FUNCTION_BLOCK FB_Base IMPLEMENTS I_Base
VAR_INPUT
END_VAR
VAR_OUTPUT
END_VAR
VAR
	{attribute 'instance-path'} 
    {attribute 'noinit'}
    {attribute 'hide'} 
    sInstancePath:		STRING(255);
	eState: 			E_Base;
	eRequest: 			E_Base;
	nState: 			INT;
	sName:				STRING(255):= 'test-run'; 	// Name OF the entire test run
	sTimestamp:			STRING(39);						// timestamp   Date and time of when the test suite was executed (in ISO 8601 format)
    {attribute 'hide'} 
	fbTask:				GETCURTASKINDEX;
	fbGetTime:			NT_GetTime;
	fCycleTime: 		LREAL;	
END_VAR

fbGetTime();

CASE eState OF
	E_Base.Init:
		IF M_Init() THEN
			eState:= E_Base.Stopped;
			nState:= 0;
		END_IF
		
	E_Base.Stopped:
		IF M_Stopped() THEN
			eState:= E_Base.Starting;
			nState:= 0;
		ELSE
			CASE eRequest OF
				E_Base.Starting, E_Base.Started:
					eState:= E_Base.Starting;
					nState:= 0;
			END_CASE
		END_IF
		
	E_Base.Starting:
		IF M_Starting() THEN
			eState:= E_Base.Started;
			nState:= 0;
		ELSE
			CASE eRequest OF
				E_Base.Started:
					eState:= E_Base.Started;
					nState:= 0;
			END_CASE
		END_IF
		
	E_Base.Started:
		IF M_Started() THEN
			eState:= E_Base.Stopping;
			nState:= 0;
		ELSE
			CASE eRequest OF
				E_Base.Stopping, E_Base.Stopped:
					eState:= E_Base.Stopping;
					nState:= 0;
			END_CASE
		END_IF
		
	E_Base.Stopping:
		IF M_Stopping() THEN
			eState:= E_Base.Stopped;
			nState:= 0;
		ELSE
			CASE eRequest OF
				E_Base.Stopped:
					eState:= E_Base.Stopped;
					nState:= 0;
			END_CASE
		END_IF
		
END_CASE

eRequest:= eState;

METHOD INTERNAL M_GetName : STRING(255)
VAR_INPUT
	sInstancePath:		STRING(255);
END_VAR
VAR
    sName:				STRING(255);
    nPosition:			INT;
END_VAR
sName := CONCAT(TwinCAT_SystemInfoVarList._AppInfo.ProjectName, '.');

nPosition := FIND(sInstancePath, sName);

IF nPosition > 0 THEN
    M_GetName:= DELETE(sInstancePath, nPosition-1 + LEN(sName), 1);
END_IF

nPosition := FIND(sInstancePath, sName);

IF nPosition > 0 THEN
    M_GetName:= DELETE(M_GetName, nPosition - 1 + LEN(sName), 1);
END_IF

nPosition:= FIND(STR1 := M_GetName, '.');
M_GetName:= RIGHT(STR := M_GetName, LEN(STR := M_GetName) - nPosition);
END_METHOD

METHOD PROTECTED M_Init : BOOL
VAR_INPUT
END_VAR
fbTask();

M_Init:= True;
END_METHOD

METHOD M_Request : BOOL
VAR_INPUT
	eState:		E_Base;
END_VAR
eRequest:= eState;
M_Request:= TRUE;
END_METHOD

METHOD PROTECTED M_Started : BOOL
VAR_INPUT
END_VAR
END_METHOD

METHOD PROTECTED M_Starting : BOOL
VAR_INPUT
END_VAR
IF fbGetTime.START THEN
	IF fbGetTime.BUSY THEN
		;
	ELSE
		sTimestamp:= SYSTEMTIME_TO_ISO8601(fbGetTime.TIMESTR, 0, FALSE, 2);
		fbGetTime.START:= FALSE;
		M_Starting:= TRUE;
	END_IF
ELSE
	sName:= M_GetName(sInstancePath);
	fCycleTime:= UDINT_TO_LREAL(TwinCAT_SystemInfoVarList._TaskInfo[fbTask.index].CycleTime) / 10000000;
	fbGetTime.START:= TRUE;
END_IF
END_METHOD

METHOD PROTECTED M_Stopped : BOOL
VAR_INPUT
END_VAR
END_METHOD

METHOD PROTECTED M_Stopping : BOOL
VAR_INPUT
END_VAR
M_Stopping:= True;
END_METHOD

PROPERTY PUBLIC P_Name : STRING(255)
GET
P_Name:= sName;
END_GET
SET
sName:= P_Name;
END_SET
END_PROPERTY

PROPERTY PUBLIC P_State : E_Base
GET
P_State:= eState;
END_GET
END_PROPERTY

END_FUNCTION_BLOCK

(* stored: Version 1.1.0.1
   POU FB_Base: Id {83180dff-a34f-4cb4-bb72-3f658f1a77bc}, SpecialFunc None
   Method M_GetName: Id {7644e4a6-816c-4e95-a1be-94a500976a8c}
   Method M_Init: Id {e2b264db-76f6-0dba-2234-6066426e6914}
   Method M_Request: Id {bfba9944-1884-04d8-1661-c3abe89f49d3}
   Method M_Started: Id {fab29306-c16a-0fb5-0321-3e286d1045b9}
   Method M_Starting: Id {bc9486fc-909d-0efe-150c-a33931b8ee19}
   Method M_Stopped: Id {fba24db4-4a8e-0338-05a4-b3761de19ee7}
   Method M_Stopping: Id {da1ded5e-11d1-08cb-1b35-69a77760c1ee}
   Property P_Name: Id {c5aac273-51f0-4149-8f97-3d72a5185d55}
   Get Get: Id {eebe96a7-e04a-4029-8470-d5af4885b0b7}
   Set Set: Id {f57ff526-3c66-4684-8e36-c365a8fe42f2}
   Property P_State: Id {d9e0f669-bd46-078f-1943-fa0edc94c5ef}
   Get Get: Id {0e5b7a2d-df5c-054a-30f6-0a2798994d9f} *)
